FUNCTION_BLOCK FB_StandardLight IMPLEMENTS ILight
VAR
	bControlValue	: BOOL;
END_VAR

METHOD M_On
P_ControlValue := TRUE;
END_METHOD

METHOD M_Off
P_ControlValue := FALSE;
END_METHOD

PROPERTY P_ControlValue : BOOL
GET
P_ControlValue := bControlValue;
END_GET
SET
bControlValue := P_ControlValue;
END_SET
END_PROPERTY

METHOD M_Execution
END_METHOD

END_FUNCTION_BLOCK

(* stored: Version 1.1.0.1, ProductVersion 3.1.0.23
   POU FB_StandardLight: Id {d28b202b-138f-4e87-a4cb-fff68407120a}
   Method M_On: Id {3eeb9c74-f481-47e5-97d9-17a1cde6a3ed}
   Method M_Off: Id {9ad83c69-c1d6-4ee0-bf07-c8cbaa7f2dbe}
   Property P_ControlValue: Id {abc02efd-3e09-45e3-b8c0-437cc4708886}
   Get Get: Id {6cd133f6-14bc-474f-bfb3-343d5412178d}
   Set Set: Id {7abefdb8-e6ff-41d9-b740-d5d20f2d1415}
   Method M_Execution: Id {fe1e585a-c63e-4fca-8243-ec2fe2e465b6} *)
